FUNCTION_BLOCK FB_OpenSourceConstructs EXTENDS TcUnit.FB_TestSuite IMPLEMENTS Vendor.I_First, I_Second
VAR
    counter : INT; (* trailing block comment stays on this line *)
    task    : TcoCore.ITcoTask;
    name    : STRING(255);
END_VAR

FOR counter := 1 TO 10 BY 2 DO
    task.Invoke();
END_FOR
{flow}

METHOD PROTECTED GetTask : TcoCore.ITcoTaskStatus
VAR_INPUT
END_VAR
GetTask := THIS^.task.Status;
END_METHOD

END_FUNCTION_BLOCK

(* stored: Version 1.1.0.1, ProductVersion 3.1.4024.12
   POU FB_OpenSourceConstructs: Id {0d2f4a66-1b3c-4e5d-8f7a-9b0c1d2e3f40}, SpecialFunc None
   Method GetTask: Id {1e3f5b77-2c4d-5f6e-9a8b-0c1d2e3f4a51} *)
